// TIA Portal V19 export
VAR_GLOBAL   // PLC tag table "D18"
   D18_Lp_EntryReq_LB301_LB302 AT %Q200.4 : Bool;   // 258SH1
   D18_Lp_SafetyReset_LB301_LB302 AT %Q200.5 : Bool;   // 258SH3
   D18_Pb_EntryReq_LB301_LB302 AT %I200.4 : Bool;   // 258SH1
   D18_Pb_SafetyReset_LB301_LB302 AT %I200.5 : Bool;   // 258SH3
   D18_Ls AT %I1200.2 : Bool;   // 200DI2 - 258BE1/R1
END_VAR
